PROGRAM MAIN
VAR
	_fb : FB_ST10; 
	_test : BOOL;
END_VAR

IF _fb._robot() THEN 
	_test:= TRUE; 
ELSE 
	_test:= FALSE; 
END_IF
_fb._tcpIp();
IF _fb._scanner() THEN 
	_test:= FALSE; 
END_IF

END_PROGRAM

(* stored: Version 1.1.0.1, ProductVersion 3.1.4024.12
   POU MAIN: Id {5a8e1327-26d3-4e43-8559-97c135f86653}, SpecialFunc None *)
